(* PLC project Generated.project, CODESYS CODESYS V3.5 SP19 Patch 1 *)
(* stored: creationDateTime 2026-09-06T13:00:42.392419, modificationDateTime 2026-09-06T13:00:42.392419 *)

(* ======================================================================= 🔌 ST_fbEncoder_HwOut — Ordres preset de sortie codeur (HwOut) ─────────────────────────────────────────────────────────────── 🎯 Rôle : Regrouper les SEULES sorties/ordres preset d'un codeur absolu EtherCAT produits par FB_Encoder vers le PDO Rx (bus sortie). 🔒 Ownership : FB_Encoder produit ce bus ; PRG_02_Acquisition le relaie vers le device. 📄 Doc métier : DOC/AF/AF_Partie-09_Fonction_Encoder_v2.4.md ======================================================================= *)
TYPE ST_fbEncoder_HwOut : STRUCT
  PresetTriggerCmd : WORD;  (* === SORTIES BUS ETHERCAT (ordres preset vers PDO Rx) === <-- [ACT] Declenchement preset vers PDO Rx *)
  CodeSeqTriggerCmd : WORD;  (* <-- [ACT] Sequence code vers PDO Rx, maintenue a 0 *)
  PresetValueOut : UDINT;  (* <-- [ACT] Valeur brute envoyee au preset *)
END_STRUCT;
END_TYPE
